// TIA Portal V19 export
VAR_GLOBAL   // PLC tag table "Decoilers_HorizRot_IO"
   DecoilersHRot_Pivot_Ls_Rest AT %I125.3 : Bool;   // 701SQ1
   DecoilersHRot_Pivot_Ls_Work AT %I125.4 : Bool;   // 701SQ2
   DecoilersHRot_Pivot_V_Rest AT %Q100.4 : Bool;   // 701YV1
   DecoilersHRot_Pivot_V_Work AT %Q100.5 : Bool;   // 701YV2
   DecoilersHRot_Rotation_V_Dec1InLine AT %Q100.2 : Bool;   // 700YV1
   DecoilersHRot_Rotation_V_Dec2InLine AT %Q100.3 : Bool;   // 700YV2
   DecoilersHRot_Pivot_Ls_ExtraMin AT %I125.1 : Bool;   // 692SQ1
   DecoilersHRot_Pivot_Ls_ExtraMax AT %I125.2 : Bool;   // 692SQ2
END_VAR
